// TIA Portal V20 export
TYPE "typeRecipe"
// stored: Access Published, Namespace Unit1
   STRUCT
      processUnitNo : Int;
      selectedRecipeTypeID : Int;
      selectedRecipeID : Int;
      currentRecipeName : WString;
      currentRecipeID : Int;
      unitRecipe : "typeUnitRecipe";
   END_STRUCT;
END_TYPE
